# EPICS substitutions: hugo/source/db/Beckhoff_9XXX/ecmcEL9576.substitutions
file "ecmcEL9576-chX.template"
{
  pattern {CH_ID}
          {01   }
}
